{attribute 'qualified_only'}
{attribute 'strict'}
TYPE E_SimStationState :
(
	IDLE := 0,
	WORKING := 1,
	DONE := 2,
	FAULTEDS := 3
);
END_TYPE

(* stored: Version 1.1.0.1, ProductVersion 3.1.4024.12
   DUT E_SimStationState: Id {015a3e3e-a22f-4b95-bec4-ccc634b591cb} *)
